FUNCTION_BLOCK FB_VFS
(* This function block implements basic functionality for Fast Shutter/Valves*)
(* Create a separate virtual PLC for the fast shutter logic, and tie/map this task to the FAST I/O portion of the ethercat bus,
 so we can scan these I/Os faster than the rest of the vacuum I/Os.
The Fast shutter was tested with PLC task Cycle Base Time 50us with cycle time 0.050ms.
*)
VAR_IN_OUT
	
END_VAR
VAR_INPUT
	{attribute 'pytmc' := 'pv: PMPS_OK'}
	i_xPMPS_OK:	BOOL	; (*External MPS interlock, Set to TRUE when no PMPS interlock is required*)
	i_xExt_OK: BOOL; (*Other External Interlock, Set to True when no external interlock is required*)
	i_xOverrideMode : BOOL; (*To be linked to global override bit. This Overrides Vacuum logic only, EPS, MPS and PMPS are still enforces*)
	// Reset fault
	{attribute 'pytmc' := '
    pv: FF_Reset
	'}
    i_xFFReset: BOOL;
END_VAR
VAR_OUTPUT
	{attribute 'pytmc' := '
    pv:
	'}
	iq_stValve : ST_VGC; (* All valve data and states will be in this struct*)
	
	
END_VAR	
VAR_IN_OUT
	io_fbFFHWO    :    FB_HardwareFFOutput;
	
END_VAR
VAR
	// PMPS
	fbFF    :    FB_FastFault :=(
        i_DevName := 'VGC',
        i_Desc := 'Fault occurs when fast sensor trips or the valve is not in open state',
        i_TypeCode := 16#1010);
	
	rDiffPressAllowed	:	REAL := 22.5; // Torr, Default value comes from Vat Valve Manual
	rDiffPress : REAL;
	set : BOOL;
    reset: BOOL;
	  
	xFirstPass	:	BOOL;
	fbFSInit		:	R_TRIG;
	
	tonDelOK : TON;
	rtOK	:	R_TRIG;
	tonOvrd	:	TON;
	
	tDelOK	:	TIME := T#60S;
	tOvrd	:	TIME := T#10s;
	
	xClose: BOOL;
	CloseTimer: TON;
	TimDur: TIME := T#20MS;
	
	(* Timeouts*)
	tTimeOutDuration: TIME:= T#0.5S;
	tOPNtimeout: TON;
	tCLStimeout:TON;
	
	
	(*IO*)
	i_xPress_OK AT%I*:BOOL; (*To be linked to the Fast sensor structure signal IG.xPRESS_OK, to make sure that the device is connected*)
	i_xOpnLS	AT%I*: BOOL;
	i_xClsLS	AT%I*: BOOL;
	q_xClose_A	AT%Q*: BOOL;
	q_xClose_B	AT%Q*: BOOL;
	q_xClose_C	AT%Q*: BOOL;
	q_xOPN_DO	AT%Q*: BOOL;
	i_xTrigger	AT%I*: BOOL; // Could be Up to 4
	q_xTrigger	AT%Q*: BOOL; // Could be Up to 4
	
	xMPS_OK	 AT%Q*:	BOOL; (*MPS Fast OK, is set when the Valve is Open and there is no trigger*)
	
	xVAC_FAULT_OK AT%Q*: BOOL; (*Valve Vacuum OK, is set to False when there is Vacuum Fault*)
	
END_VAR

//TODO
// Make it better
//Test It
//Fix PVs and IO links
//Interface with neighboring valves.
//PMPS requirement ??

(* Fast Shutter/Valve Function Block*)
(* M.Ghaly Feb 2019*)

(* Fast Shutters do not function as complete isolation valves, but are intended to rapidly limit conductance 
between vacuum regions.  They should be installed in conjunction with isolation gate valves.  The conductance 
of the fast shutter in the closed state may be sufficiently low as to create an isolated vacuum region.  
Thus, at least a pirani gauge, that can measure a pressure down to 1x10-4 Torr, needs to be installed between
the shutter and the isolation gate valve.
In the case where a gauge is not installed, the neigboring gate Valves should not be opened unless the shutter 
is Open. 
*)
(* Soft IO Mapping*)
IO();

///Check valve postion
IF iq_stValve.i_xClsLS AND  iq_stValve.i_xOpnLS THEN
	iq_stValve.eState:=INVALID;
ELSIF NOT iq_stValve.i_xClsLS AND iq_stValve.i_xOpnLS AND iq_stValve.q_xOPN_DO THEN 
	iq_stValve.eState:=OPEN;
ELSIF iq_stValve.i_xClsLS AND NOT iq_stValve.i_xOpnLS AND NOT iq_stValve.q_xOPN_DO THEN 
	iq_stValve.eState:=CLOSED;
ELSIF NOT iq_stValve.i_xClsLS AND NOT iq_stValve.i_xOpnLS THEN 
	iq_stValve.eState:=MOVING;
ELSE
	iq_stValve.eState:=INVALID;
END_IF

(* Input Trigger to close the Fast Shutter*)
(* Neighboring Valves Should also be triggered to Close*)
IF (i_xTrigger) OR NOT (i_xPress_OK) OR NOT (i_xExt_OK)  OR NOT (iq_stValve.pv_xOPN_SW)  THEN 
	xClose:= TRUE;
	iq_stValve.pv_xOPN_SW := FALSE;
	xVAC_FAULT_OK:= FALSE;
	iq_stValve.xERR_ExtFault := TRUE;
END_IF
IF (xClose) AND (NOT i_xClsLS) THEN
	q_xClose_A := TRUE;
	q_xClose_B := TRUE;
	q_xClose_C := TRUE;
END_IF
IF(CloseTimer.Q) OR (i_xClsLS) THEN
	q_xClose_A := FALSE;
	q_xClose_B := FALSE;
	q_xClose_C := FALSE;
	xClose := FALSE;
	iq_stValve.pv_xOPN_SW := FALSE;
END_IF

(* Neighboring Valves Interlock bit is reset When the Vacuum event error is reset and the Shutter is opened *)
IF (NOT i_xTrigger) AND (NOT iq_stValve.xERR_ExtFault) AND i_xOpnLS THEN
	xVAC_FAULT_OK := TRUE;
END_IF

(*OPN OK evaluation bit *)
iq_stValve.xOPN_OK := (NOT iq_stValve.xERR_ExtFault) AND NOT i_xTrigger;

(* If Epics Command to close the Valve, check if PMPS, otherwise Keep command set to open valve *)
// is there really a PMPS requirment.



(* Here's where the valve opens *)
iq_stValve.q_xOPN_DO := (iq_stValve.pv_xOPN_SW AND iq_stValve.xOPN_OK) OR (tonOvrd.Q AND i_xOverrideMode);

(* When the valve  is open MPS is OK*)
xMPS_OK := (iq_stValve.eState=OPEN) AND NOT i_xTrigger AND i_xPress_OK;//gauge is connected


(* Override logic *)
(* Goal: give ability to override, but do so in a way that people won't forget it.
Solution: Override only after ten seconds of override, protect against blips,
when the valve permission goes true for more than ten seconds consistently, remove override
*)

tonDelOK(IN:=iq_stValve.xOPN_OK, PT:=tDelOK);
rtOK(CLK:=tonDelOK.Q);
IF rtOK.Q AND iq_stValve.pv_xOvrdOpn THEN 
	iq_stValve.pv_xOvrdOpn :=FALSE;
	iq_stValve.pv_xOPN_SW := TRUE; //for seamless transition
END_IF

//Override timer
tonOvrd(IN:=iq_stValve.pv_xOvrdOpn, PT:=tOvrd);



///Check valve postion timout
IF NOT iq_stValve.i_xClsLS AND tCLStimeout.Q THEN 
	iq_stValve.bErrorPresent := TRUE;
ELSIF NOT iq_stValve.i_xOpnLS AND tOPNtimeout.Q THEN 
	iq_stValve.bErrorPresent := TRUE;
END_IF

(*Timers*)
CloseTimer ( IN:=xClose, PT:= TimDur, Q=>);
tOPNtimeout(IN:= iq_stValve.q_xOPN_DO, PT := tTimeOutDuration );
tCLStimeout(IN:= NOT iq_stValve.q_xOPN_DO, PT := tTimeOutDuration);

(* Soft IO Mapping*)
IO();
// Alarm reset
//////////////////////////////////////
ACT_ResetAlarms();


(*FAST FAULT*)
fbFF(i_xOK := xMPS_OK,
    i_xReset := i_xFFReset,
    io_fbFFHWO := io_fbFFHWO);

ACTION ACT_ResetAlarms:
iq_stValve.xERR_DifPres R= iq_stValve.pv_xAlmRst;

iq_stValve.bErrorPresent R= iq_stValve.pv_xAlmRst;

IF NOT i_xTrigger THEN
	iq_stValve.xERR_ExtFault R= iq_stValve.pv_xAlmRst;
END_IF
END_ACTION

ACTION IO:
(*inputs*)
iq_stValve.i_xOpnLS := 	i_xOpnLS;
iq_stValve.i_xClsLS:=	i_xClsLS;
iq_stValve.xEXT_OK := i_xEXT_OK;
iq_stValve.xOverrideMode := i_xOverrideMode;
(*outputs*)
q_xOPN_DO:= iq_stValve.q_xOPN_DO;
q_xTrigger:=i_xTrigger;
END_ACTION

END_FUNCTION_BLOCK

(* stored: Version 1.1.0.1, ProductVersion 3.1.4022.16
   POU FB_VFS: Id {68519563-003c-4daf-ae0e-7245b1fe09af}, SpecialFunc None
   Action ACT_ResetAlarms: Id {5bc381e2-d93d-4e07-9868-4d1094f97e97}
   Action IO: Id {be2b8137-473d-4278-9e2c-831399c62f45} *)
